// LS Electric XG5000 project: modbus
// PLC LSPLC
// module base 0 slot 0: 입출력 모듈:XBC-DR14E (DC 24V 입력 8점, 릴레이 출력 6점)

PROGRAM NewProgram (task: 스캔 프로그램)

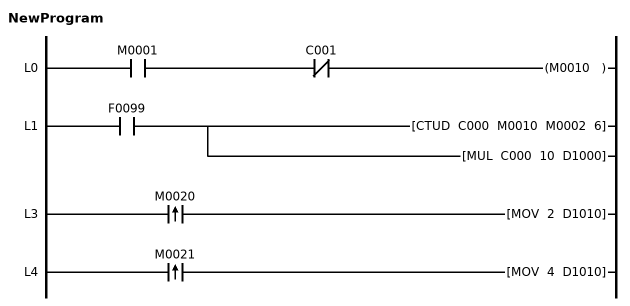
; L0
LOAD      M0001
AND NOT   C001
OUT       M0010
; L1
LOAD      F0099
CTUD      C000 M0010 M0002 6
MUL       C000 10 D1000
; L3
LOADP     M0020
MOV       2 D1010
; L4
LOADP     M0021
MOV       4 D1010